// Mitsubishi GX Works2 project: PLC_GROUP25_20_04   PLC: FX3G

// global labels: Global1
VAR_GLOBAL
  switch3 AT X003 : BOOL;  (* empty_mold_sensor / משתנה זה מייצג את חיישן המיקום X3, מזהה סט תבניות ריקות ומתחיל את תהליך היציקה, יכול לקבל ערך 0 או 1. *)
  TS_1 AT TS1 : BOOL;  (* casting_process_complete / המשתנה הזה מקבל ערך 1 בסוף תהליך היציקה, מציין את סיום התהליך. *)
  light2 AT Y002 : BOOL;  (* casting_indicator_light / המשתנה הזה דולק בזמן היציקה ומייצג אינדיקטור לכך שתהליך היציקה מתרחש. *)
  TC_1 AT TC1 : BOOL;  (* casting_timer / המשתנה הזה מייצג את הטיימר של תהליך היציקה. *)
END_VAR
VAR_GLOBAL CONSTANT
  Yetzka_time : INT := 40;  (* CASTING_TIME_CONSTANT / משתנה הזה הוא קבוע שמייצג את זמן היציקה, עם ערך קבוע של 40. *)
END_VAR
VAR_GLOBAL
  switch1 AT X001 : BOOL;  (* melting_start_button / המשתנה הזה מייצג את כפתור תחילת ההמסה, יכול לקבל ערך 0 או 1. *)
END_VAR
VAR_GLOBAL CONSTANT
  Pass_choc : REAL := 400;  (* CHOCOLATE_PER_BATCH_CONSTANT / המשתנה הזה הוא קבוע שמסמן את כמות השוקולד במנת ייצור אחת. *)
END_VAR
VAR_GLOBAL
  switch2 AT X002 : BOOL;  (* temperature_threshold_sensor / המשתנה הזה מייצג כפתור שמסמן חיישן, נותן ערך 1 כאשר הטמפרטורה מגיעה ל-45 מעלות. *)
  light1 AT Y001 : BOOL;  (* melting_indicator_light / המשתנה הזה דולק בזמן ההמסה ומסמן שתהליך ההמסה מתרחש. *)
  switch4 AT X004 : BOOL;  (* filling_process_start_button / המשתנה הזה מייצג את כפתור תחילת תהליך המילוי. משתנה הזה מייצג את כפתור תחילת תהליך המילוי - יכול לקבל 0 או 1 *)
  Nunts_Mix AT M100 : BOOL;  (* nut_chocolate_selection / משתנה עזר שמקבל ערך 1 אם נבחר שוקולד אגוזים ו-0 אם נבחר שוקולד דובאי. *)
  saved_analogInput1 AT D1111 : INT;  (* saved_analogInput1 / רגיסטר אליו מעבירים את הערך שקיבלנו מהרגיסטר עם הערך האנלוגי. *)
  move_m AT M1 : BOOL;  (* move_m / אינדיקטור שמקבל ערך 1 לאחר ביצוע העברת הערך מהרגיסטר האנלוגי. *)
END_VAR
VAR_GLOBAL CONSTANT
  const_5 : INT := 5;
END_VAR
VAR_GLOBAL
  light3 AT Y003 : BOOL;  (* filling_process_indicator_light1 / מהבהב בזמן ביצוע תהליך המילוי, מציין שהתהליך פעיל. *)
  light4 AT Y004 : BOOL;  (* filling_process_indicator_light2 / מהבהב בזמן ביצוע תהליך המילוי, מציין שהתהליך פעיל. *)
END_VAR
VAR_GLOBAL CONSTANT
  Fist_num_dubai : REAL := 120;  (* פיסטוק *)
  Kad_num_dubai : REAL := 60;  (* קדאיף *)
END_VAR
VAR_GLOBAL
  finish_moving AT M2 : BOOL;
END_VAR
VAR_GLOBAL CONSTANT
  Nut_num_Nuts : REAL := 100;  (* אגוזים *)
  Fist_num_nuts : REAL := 100;  (* פיסטוק *)
END_VAR
VAR_GLOBAL
  TC_2 AT TC2 : BOOL;
  TS_2 AT TS2 : BOOL;
END_VAR
VAR_GLOBAL CONSTANT
  const_50 : INT := 50;
END_VAR
VAR_GLOBAL
  m_3 AT M3 : BOOL;
  TC_3 AT TC3 : BOOL;
  TS_3 AT TS3 : BOOL;
  TC_4 AT TC4 : BOOL;
  TS_4 AT TS4 : BOOL;
  switch6 AT X006 : BOOL;  (* cooling *)
  TC_5 AT TC5 : BOOL;
END_VAR
VAR_GLOBAL CONSTANT
  const_30 : INT := 30;
END_VAR
VAR_GLOBAL
  TS_5 AT TS5 : BOOL;
  light6 AT Y006 : BOOL;
  switch0 AT X000 : BOOL;
  storage AT D1113 : REAL;
  CC_1 AT CC1 : BOOL;
END_VAR
VAR_GLOBAL CONSTANT
  const_4 : INT := 4;
END_VAR
VAR_GLOBAL
  light5 AT Y005 : BOOL;
  CS_1 AT CS1 : BOOL;
END_VAR
VAR_GLOBAL CONSTANT
  const_1 : REAL := 1;
END_VAR
VAR_GLOBAL
  holding_3 AT M4 : BOOL;
  Check_Term AT M5 : BOOL;
  indicator1 AT M6 : BOOL;
  indicator2 AT M7 : BOOL;
  indicator3 AT M8 : BOOL;
  indicator4 AT M9 : BOOL;
  stock_not_ok AT M11 : BOOL;
  light7 AT Y007 : BOOL;
  switch5 AT X005 : BOOL;
  indicator5 AT M12 : BOOL;
  indicator6 AT M13 : BOOL;
END_VAR
VAR_GLOBAL CONSTANT
  const_10 : REAL := 10;
END_VAR
VAR_GLOBAL
  ChockNum_ORGINIAL AT D7998 : REAL;  (* כמות שוקולד מקורית *)
  Nut_num_ORGINIAL AT D7996 : REAL;  (* אגוזים כמות מקורית *)
  Fist_num_ORGINIAL AT D7994 : REAL;  (* כמות שוקולד מקורית *)
  Kad_num_ORGINIAL AT D7992 : REAL;  (* אגוזים כמות מקורית *)
  temp : REAL;
END_VAR
VAR_GLOBAL CONSTANT
  const_0 : REAL;
END_VAR
VAR_GLOBAL
  tetempmp : WORD;
  saved_analogInput2 AT D8201 : REAL;
  analogInput1 AT D8280 : INT;
END_VAR
VAR_GLOBAL CONSTANT
  const_400 : REAL := 400;
  storage1 : INT := 80;
END_VAR
VAR_GLOBAL
  analogoutput AT D8282 : INT;
END_VAR
VAR_GLOBAL CONSTANT
  const_00 : INT;
END_VAR
VAR_GLOBAL
  indicator12 AT M19 : BOOL;  (* נדלק כשמסיימים את ההעמסה *)
  indicator13 AT M20 : BOOL;
  indicator14 AT M21 : BOOL;
END_VAR
VAR_GLOBAL CONSTANT
  Nut_num_dubai : REAL := 20;  (* dubai_chocolate_nut_quantity_constant / קבוע שמסמל את כמות האגוזים שצריך לשים בשוקולד דובאי. *)
END_VAR
VAR_GLOBAL
  switch7 AT X007 : BOOL;
  ChockNum AT D1100 : REAL;  (* chocolate_inventory_quantity / המשתנה הזה מייצג את כמות השוקולד במלאי, מאוכסן כערך עשרוני (רגיסטר). *)
  Nut_num AT D1103 : REAL;  (* nut_quantity / רגיסטר - המייצג את מלאי האגוזים הנוכחי *)
  Fist_num AT D1106 : REAL;  (* פיסטוק *)
  Kad_num AT D1109 : REAL;  (* שערות קדאיף *)
END_VAR

// task Task_01 (event TRUE, interval 0, priority 31): POU_01

PROGRAM POU_01
(* structured ladder/FBD written out as ST: instructions are called as NAME(EN, inputs, outputs); _pN, _eN, _tN stand for wires *)
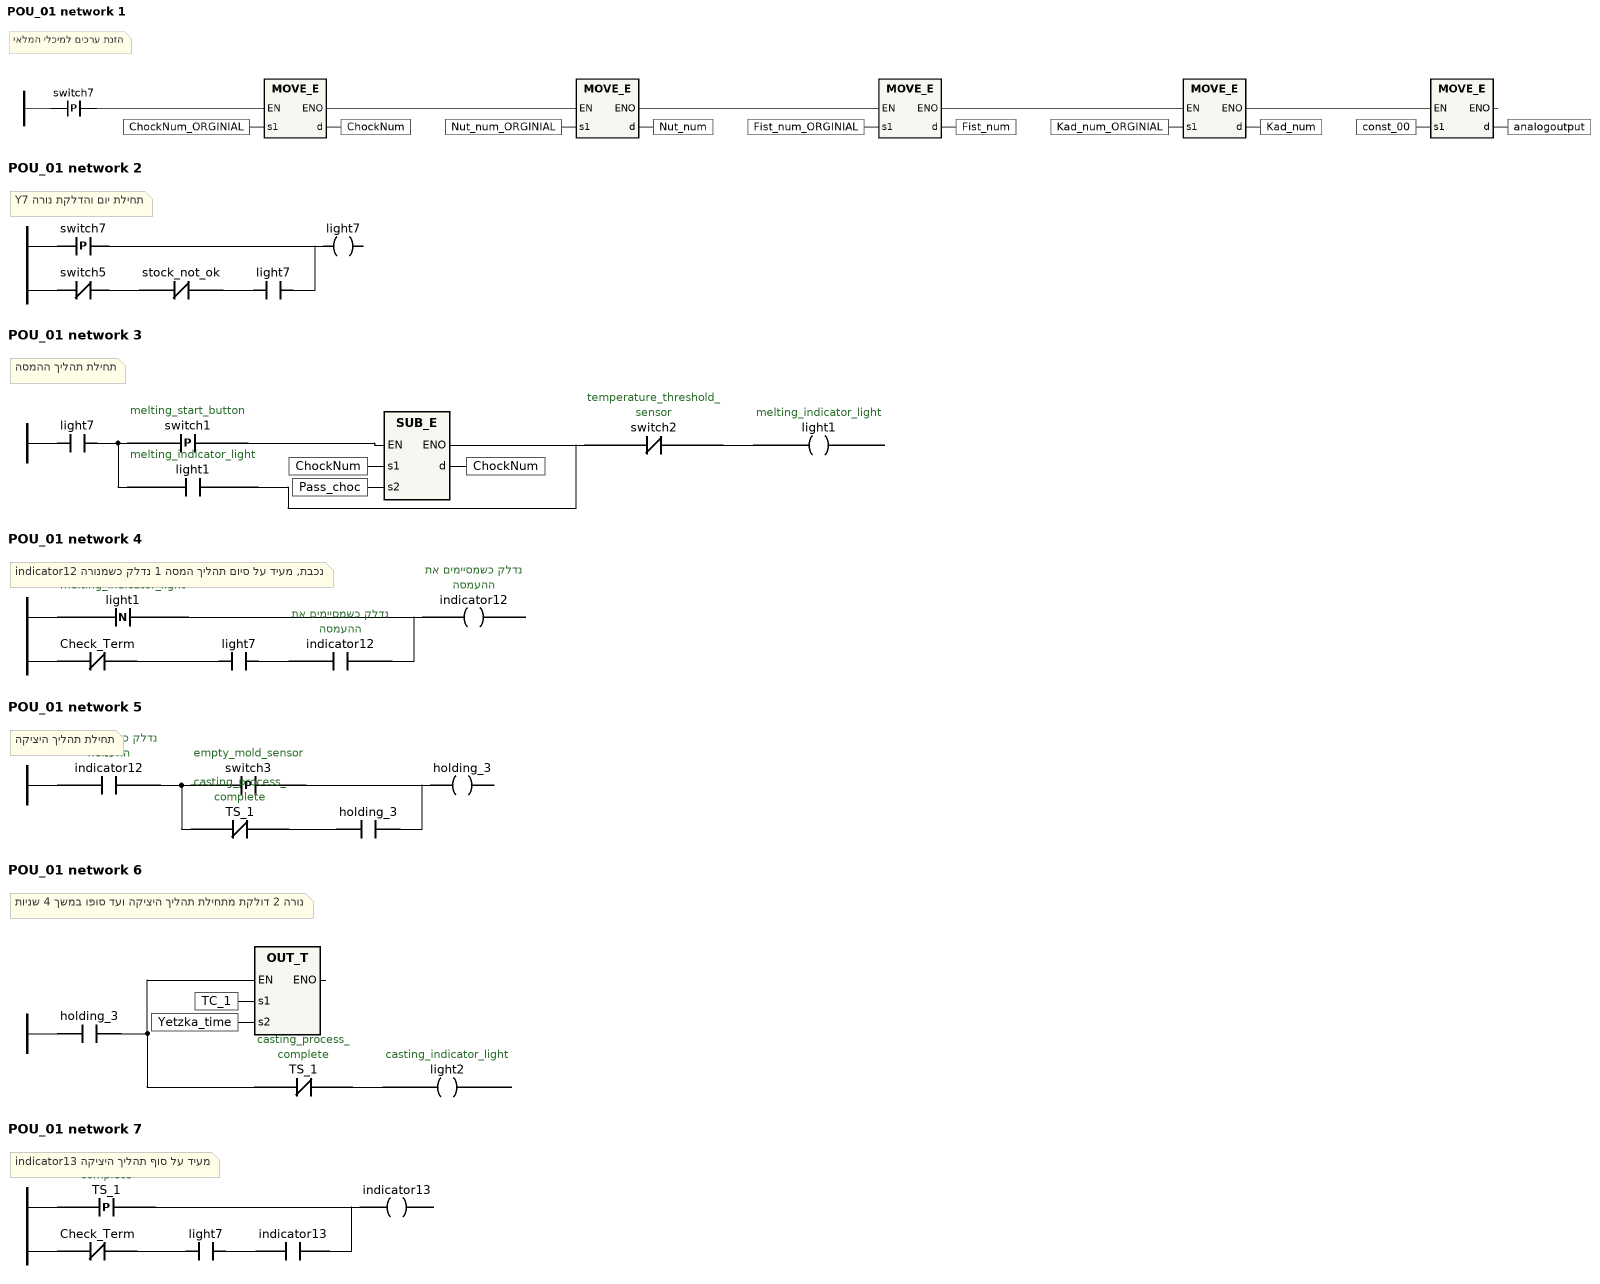
(* network 1 *)
(* הזנת ערכים למיכלי המלאי *)
_e1 := MOVE_E(LDP(TRUE, switch7), ChockNum_ORGINIAL, ChockNum);
_e2 := MOVE_E(_e1, Nut_num_ORGINIAL, Nut_num);
_e3 := MOVE_E(_e2, Fist_num_ORGINIAL, Fist_num);
_e4 := MOVE_E(_e3, Kad_num_ORGINIAL, Kad_num);
MOVE_E(_e4, const_00, analogoutput);
(* network 2 *)
(* תחילת יום והדלקת נורה Y7 *)
light7 := LDP(TRUE, switch7) OR (NOT switch5 AND NOT stock_not_ok AND light7);
(* network 3 *)
(* תחילת תהליך ההמסה *)
_e1 := SUB_E(light7 AND LDP(TRUE, switch1), ChockNum, Pass_choc, ChockNum);
light1 := (_e1 OR (light7 AND light1)) AND NOT switch2;
(* network 4 *)
(* indicator12 נדלק כשמנורה 1 נכבת, מעיד על סיום תהליך המסה *)
indicator12 := LDF(TRUE, light1) OR (NOT Check_Term AND light7 AND indicator12);
(* network 5 *)
(* תחילת תהליך היציקה *)
holding_3 := (indicator12 AND LDP(TRUE, switch3)) OR (indicator12 AND NOT TS_1 AND holding_3);
(* network 6 *)
(* נורה 2 דולקת מתחילת תהליך היציקה ועד סופו במשך 4 שניות *)
OUT_T(holding_3, TC_1, Yetzka_time);
light2 := holding_3 AND NOT TS_1;
(* network 7 *)
(* indicator13 מעיד על סוף תהליך היציקה *)
indicator13 := LDP(TRUE, TS_1) OR (NOT Check_Term AND light7 AND indicator13);
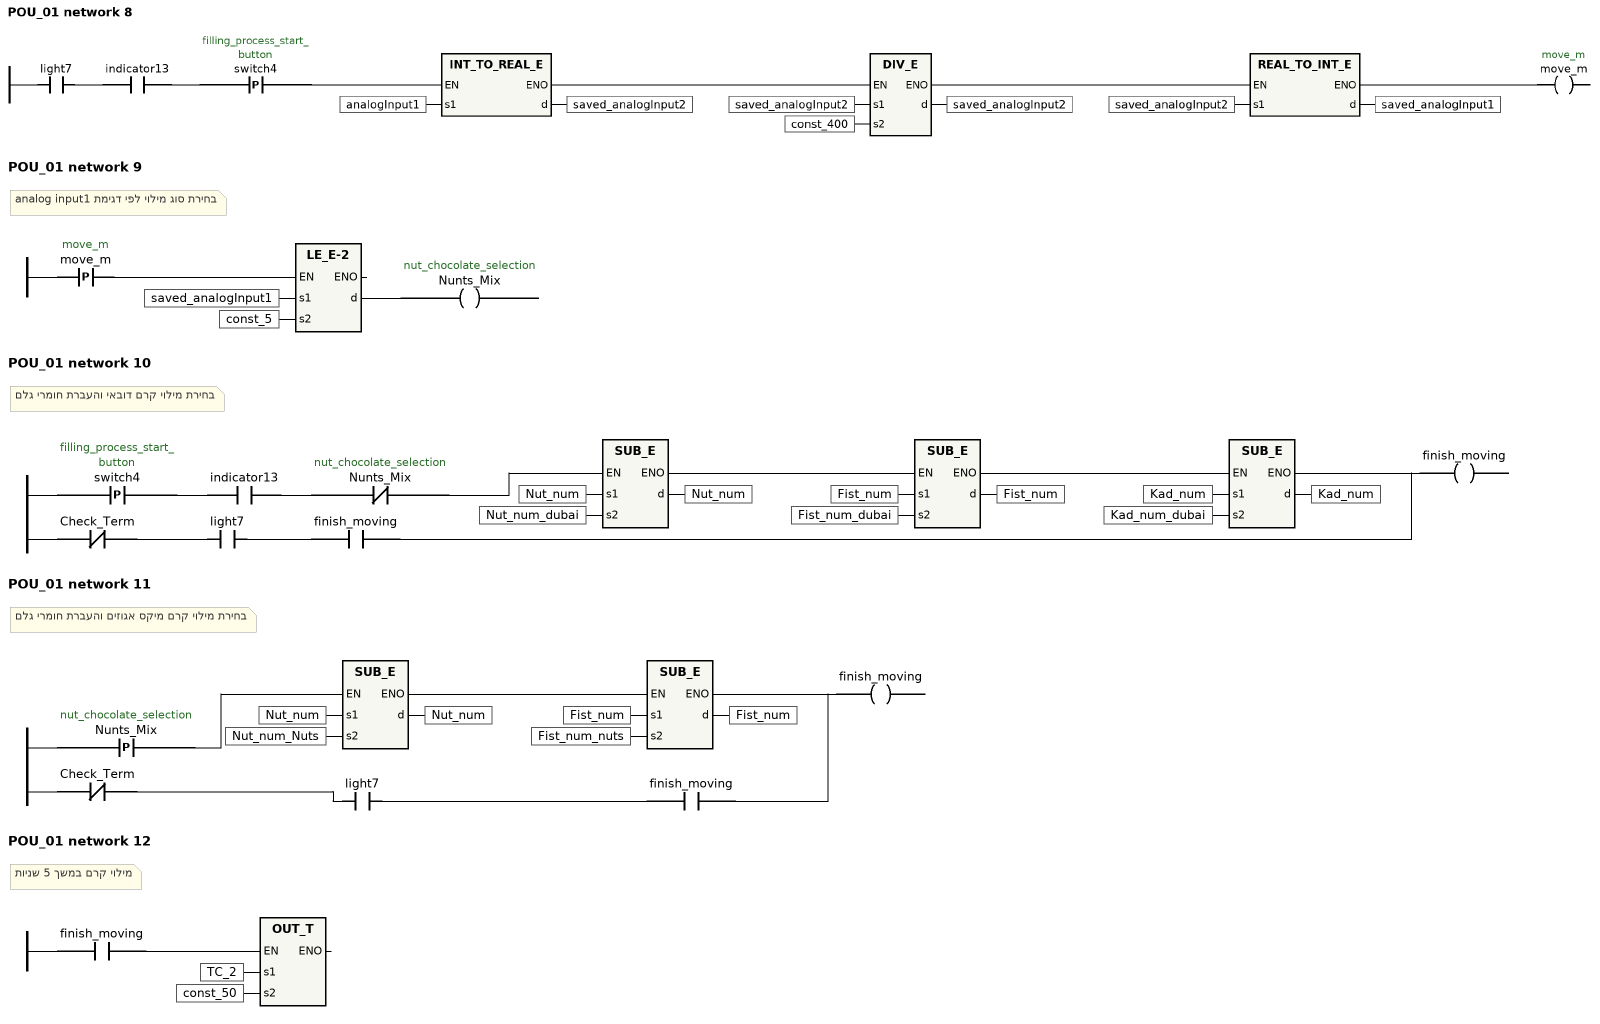
(* network 8 *)
_e1 := INT_TO_REAL_E(light7 AND indicator13 AND LDP(TRUE, switch4), analogInput1, saved_analogInput2);
_e2 := DIV_E(_e1, saved_analogInput2, const_400, saved_analogInput2);
_e3 := REAL_TO_INT_E(_e2, saved_analogInput2, saved_analogInput1);
move_m := _e3;
(* network 9 *)
(* בחירת סוג מילוי לפי דגימת analog input1 *)
LE_E(LDP(TRUE, move_m), saved_analogInput1, const_5, _t1);
Nunts_Mix := _t1;
(* network 10 *)
(* בחירת מילוי קרם דובאי והעברת חומרי גלם *)
_e1 := SUB_E(LDP(TRUE, switch4) AND indicator13 AND NOT Nunts_Mix, Nut_num, Nut_num_dubai, Nut_num);
_e2 := SUB_E(_e1, Fist_num, Fist_num_dubai, Fist_num);
_e3 := SUB_E(_e2, Kad_num, Kad_num_dubai, Kad_num);
finish_moving := _e3 OR (NOT Check_Term AND light7 AND finish_moving);
(* network 11 *)
(* בחירת מילוי קרם מיקס אגוזים והעברת חומרי גלם *)
_e1 := SUB_E(LDP(TRUE, Nunts_Mix), Nut_num, Nut_num_Nuts, Nut_num);
_e2 := SUB_E(_e1, Fist_num, Fist_num_nuts, Fist_num);
finish_moving := _e2 OR (NOT Check_Term AND light7 AND finish_moving);
(* network 12 *)
(* מילוי קרם במשך 5 שניות *)
OUT_T(finish_moving, TC_2, const_50);
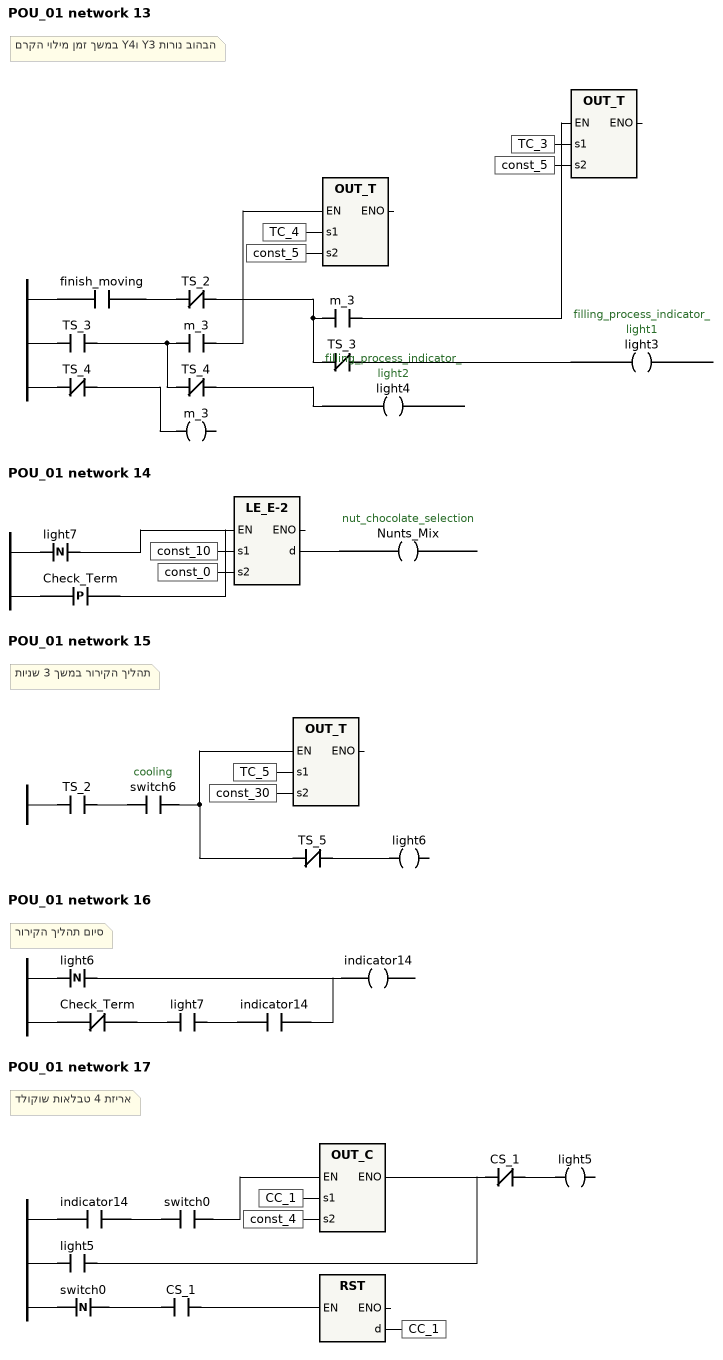
(* network 13 *)
(* הבהוב נורות Y3 וY4 במשך זמן מילוי הקרם *)
_p1 := finish_moving AND NOT TS_2;
OUT_T(_p1 AND m_3, TC_3, const_5);
light3 := _p1 AND NOT TS_3;
OUT_T(TS_3 AND m_3, TC_4, const_5);
light4 := TS_3 AND NOT TS_4;
m_3 := NOT TS_4;
(* network 14 *)
LE_E(LDF(TRUE, light7) OR LDP(TRUE, Check_Term), const_10, const_0, _t1);
Nunts_Mix := _t1;
(* network 15 *)
(* תהליך הקירור במשך 3 שניות *)
_p1 := TS_2 AND switch6;
OUT_T(_p1, TC_5, const_30);
light6 := _p1 AND NOT TS_5;
(* network 16 *)
(* סיום תהליך הקירור *)
indicator14 := LDF(TRUE, light6) OR (NOT Check_Term AND light7 AND indicator14);
(* network 17 *)
(* אריזת 4 טבלאות שוקולד *)
_e1 := OUT_C(indicator14 AND switch0, CC_1, const_4);
light5 := (_e1 OR light5) AND NOT CS_1;
RST(LDF(TRUE, switch0) AND CS_1, CC_1);
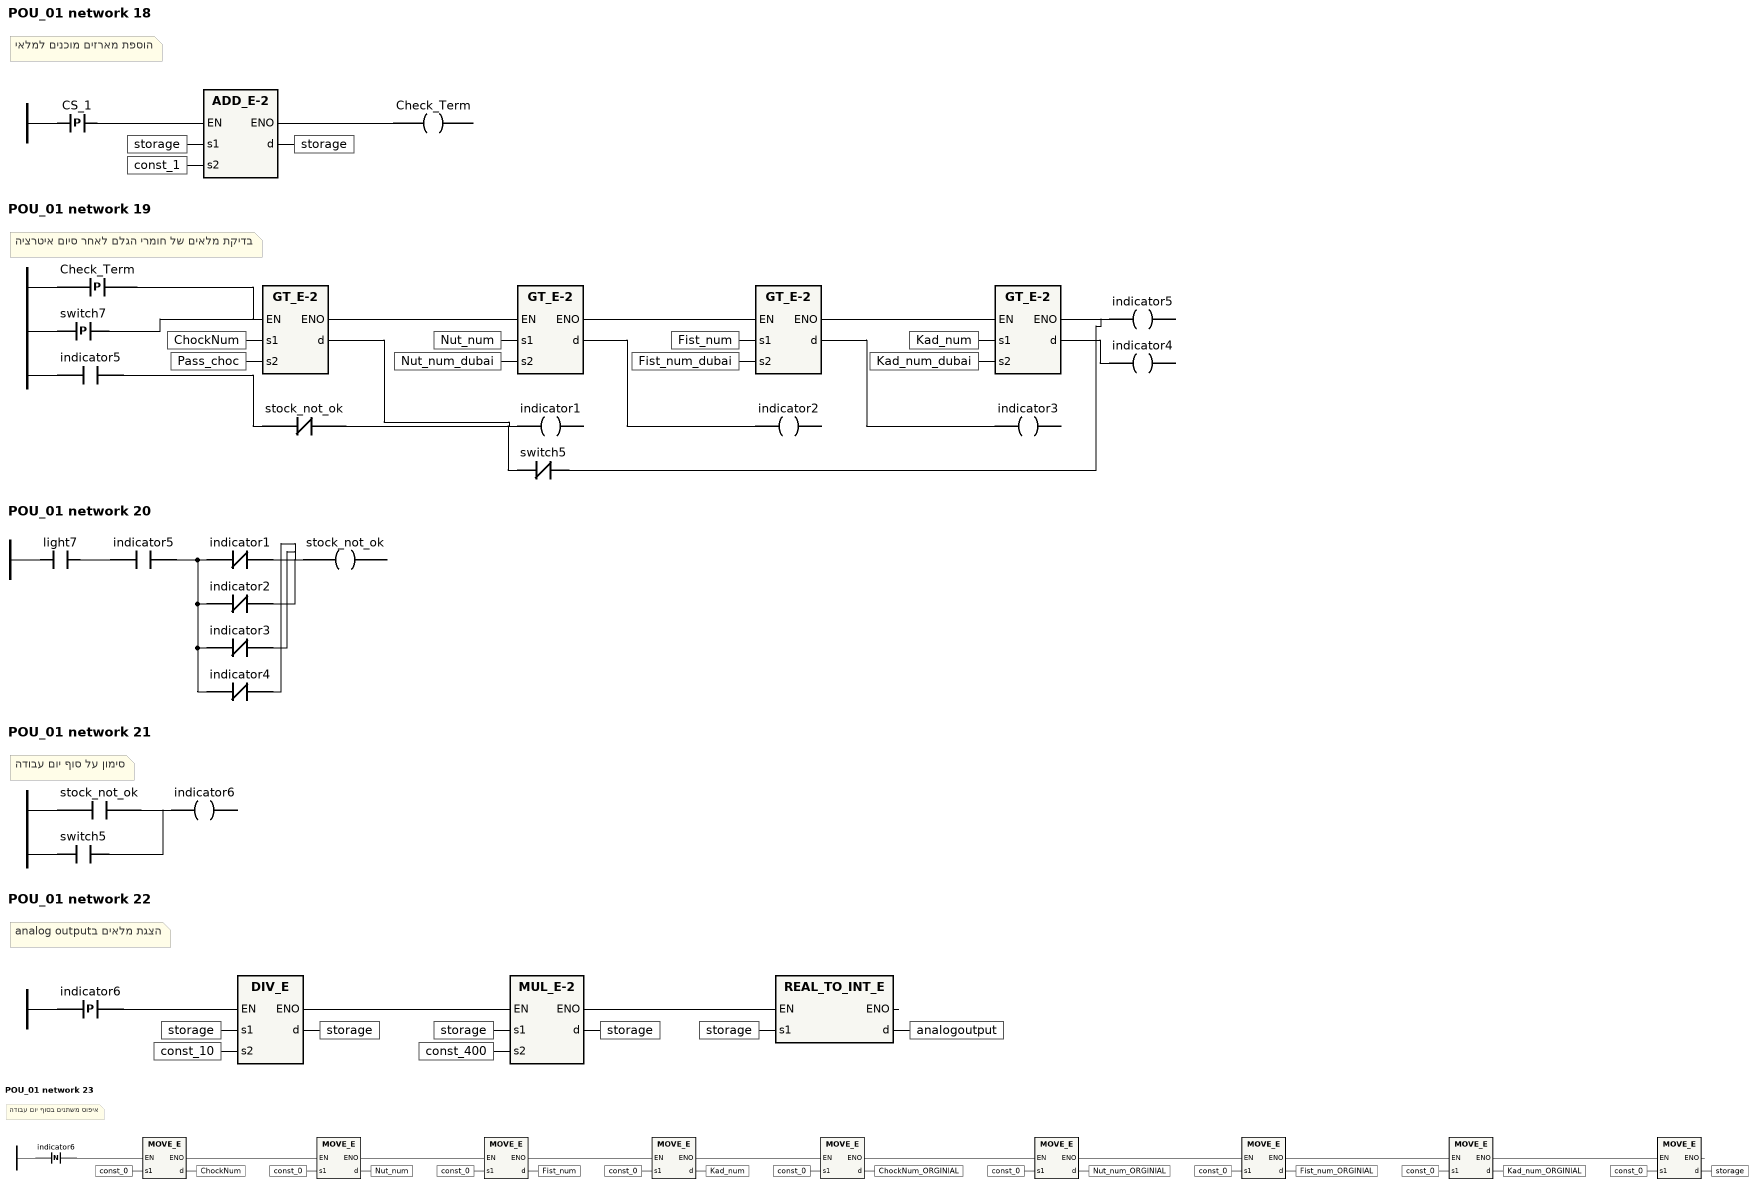
(* network 18 *)
(* הוספת מארזים מוכנים למלאי *)
_e1 := ADD_E(LDP(TRUE, CS_1), storage, const_1, storage);
Check_Term := _e1;
(* network 19 *)
(* בדיקת מלאים של חומרי הגלם לאחר סיום איטרציה *)
_e2 := GT_E(LDP(TRUE, Check_Term) OR LDP(TRUE, switch7), ChockNum, Pass_choc, _t1);
_e4 := GT_E(_e2, Nut_num, Nut_num_dubai, _t3);
_e6 := GT_E(_e4, Fist_num, Fist_num_dubai, _t5);
_e8 := GT_E(_e6, Kad_num, Kad_num_dubai, _t7);
indicator5 := _e8 OR (indicator5 AND NOT stock_not_ok AND NOT switch5);
indicator1 := _t1;
indicator2 := _t3;
indicator3 := _t5;
indicator4 := _t7;
(* network 20 *)
_p1 := light7 AND indicator5;
stock_not_ok := (_p1 AND NOT indicator1) OR (_p1 AND NOT indicator2) OR (_p1 AND NOT indicator3) OR (_p1 AND NOT indicator4);
(* network 21 *)
(* סימון על סוף יום עבודה *)
indicator6 := stock_not_ok OR switch5;
(* network 22 *)
(* הצגת מלאים בanalog output *)
_e1 := DIV_E(LDP(TRUE, indicator6), storage, const_10, storage);
_e2 := MUL_E(_e1, storage, const_400, storage);
REAL_TO_INT_E(_e2, storage, analogoutput);
(* network 23 *)
(* איפוס משתנים בסוף יום עבודה *)
_e1 := MOVE_E(LDF(TRUE, indicator6), const_0, ChockNum);
_e2 := MOVE_E(_e1, const_0, Nut_num);
_e3 := MOVE_E(_e2, const_0, Fist_num);
_e4 := MOVE_E(_e3, const_0, Kad_num);
_e5 := MOVE_E(_e4, const_0, ChockNum_ORGINIAL);
_e6 := MOVE_E(_e5, const_0, Nut_num_ORGINIAL);
_e7 := MOVE_E(_e6, const_0, Fist_num_ORGINIAL);
_e8 := MOVE_E(_e7, const_0, Kad_num_ORGINIAL);
MOVE_E(_e8, const_0, storage);
END_PROGRAM
